(* CODESYS project PacFramwork.project
   Version: 0.0.0.0
   Title: PacFramwork
   Author: roma_mirkevich

Project tree, tasks and I/O mapping:
  PacFramwork : TM241CEC24T/U, Schneider Electric, order no. TM241CEC24T/U, version 5.1.10.10
    application Application
      libraries: SysTimeRtc, * (System); SysTimeCore, * (System); CmpIecTask, * (System); CmpApp, * (System)
      task MAST (freewheeling, priority 15, watchdog 500 ms x 1) calls SR_Main
      program SR_Main [ST]
      global variables SYS
      global variables TEST
      function block PLCFN [ST]
      function TS_PLCFN [ST]
      global variables BUF
      global variables CH
      global variables HMI
      UTD/
        data type PLC_STA
        data type PLC_ALM1
        data type PLS
        data type PLC_CFG
        data type CHBUF
        data type CHCFG
        data type CHHMI
        data type CHSTA
        data type MODULE
        data type SUBMODULE
      CH/
        function CHAIFN [ST]
        function CHAOFN [ST]
        function CHDIFN [ST]
        function CHDOFN [ST]
        function MODULES [ST]
      function INPUT [ST]
      function OUTPUT [ST]
      function ACTUATOR [ST]
      global variables IO
    Ethernet_1 : Ethernet Network, Schneider Electric, version 5.1.10.10
        settings: FTP Server = false
    Serial_Line_1 : Serial line, Schneider Electric, version 5.1.10.10
      Machine_Expert_Network_Manager : Machine Expert-Network Manager, Schneider Electric, version 4.0.0.4
    Serial_Line_2 : Serial line, Schneider Electric, version 5.1.10.10
      Modbus_Manager : Modbus Manager, Schneider Electric, version 4.0.0.4
    CAN_1 : CANopen bus, Schneider Electric, version 5.1.10.10
    DI : Digital Inputs, Schneider Electric, version 5.1.10.10
        input  iwDI_IW0 : WORD  // IW0
        input  ibDI_IB1 : BYTE  // IB1
    DQ : Digital Outputs, Schneider Electric, version 5.1.10.10
        output qwDQ_QW0 : WORD  // QW0
        output qbDQ_QB1 : BYTE  // QB1
    Counters : Counters, Schneider Electric, version 5.1.10.10
    Pulse_Generators : Pulse Generators, Schneider Electric, version 5.1.10.10
    IO_Bus : IO bus - TM3, Schneider Electric, version 5.1.10.10
      Module_2 : TM3DI32K, Schneider Electric, order no. TM3DI32K, version 1.0.2.2
          input  Application.IO.DI[1] : BOOL  // ID0.I0
          input  Application.IO.DI[2] : BOOL  // ID0.I1
          input  Application.IO.DI[3] : BOOL  // ID0.I2
          input  Application.IO.DI[4] : BOOL  // ID0.I3
          input  Application.IO.DI[5] : BOOL  // ID0.I4
          input  Application.IO.DI[6] : BOOL  // ID0.I5
          input  Application.IO.DI[7] : BOOL  // ID0.I6
          input  Application.IO.DI[8] : BOOL  // ID0.I7
          input  Application.IO.DI[9] : BOOL  // ID0.I8
          input  Application.IO.DI[10] : BOOL  // ID0.I9
          input  Application.IO.DI[11] : BOOL  // ID0.I10
          input  Application.IO.DI[12] : BOOL  // ID0.I11
          input  Application.IO.DI[13] : BOOL  // ID0.I12
          input  Application.IO.DI[14] : BOOL  // ID0.I13
          input  Application.IO.DI[15] : BOOL  // ID0.I14
          input  Application.IO.DI[16] : BOOL  // ID0.I15
          input  Application.IO.DI[17] : BOOL  // ID0.I16
          input  Application.IO.DI[18] : BOOL  // ID0.I17
          input  Application.IO.DI[19] : BOOL  // ID0.I18
          input  Application.IO.DI[20] : BOOL  // ID0.I19
          input  Application.IO.DI[21] : BOOL  // ID0.I20
          input  Application.IO.DI[22] : BOOL  // ID0.I21
          input  Application.IO.DI[23] : BOOL  // ID0.I22
          input  Application.IO.DI[24] : BOOL  // ID0.I23
          input  Application.IO.DI[25] : BOOL  // ID0.I24
          input  Application.IO.DI[26] : BOOL  // ID0.I25
          input  Application.IO.DI[27] : BOOL  // ID0.I26
          input  Application.IO.DI[28] : BOOL  // ID0.I27
          input  Application.IO.DI[29] : BOOL  // ID0.I28
          input  Application.IO.DI[30] : BOOL  // ID0.I29
          input  Application.IO.DI[31] : BOOL  // ID0.I30
          input  Application.IO.DI[32] : BOOL  // ID0.I31
          unmapped channels: ID0
      Module_3 : TM3DQ32TK, Schneider Electric, order no. TM3DQ32TK, version 1.0.2.2
          output Application.IO.DQ[1] : BOOL  // QD0.Q0
          output Application.IO.DQ[2] : BOOL  // QD0.Q1
          output Application.IO.DQ[3] : BOOL  // QD0.Q2
          output Application.IO.DQ[4] : BOOL  // QD0.Q3
          output Application.IO.DQ[5] : BOOL  // QD0.Q4
          output Application.IO.DQ[6] : BOOL  // QD0.Q5
          output Application.IO.DQ[7] : BOOL  // QD0.Q6
          output Application.IO.DQ[8] : BOOL  // QD0.Q7
          output Application.IO.DQ[9] : BOOL  // QD0.Q8
          output Application.IO.DQ[10] : BOOL  // QD0.Q9
          output Application.IO.DQ[11] : BOOL  // QD0.Q10
          output Application.IO.DQ[12] : BOOL  // QD0.Q11
          output Application.IO.DQ[13] : BOOL  // QD0.Q12
          output Application.IO.DQ[14] : BOOL  // QD0.Q13
          output Application.IO.DQ[15] : BOOL  // QD0.Q14
          output Application.IO.DQ[16] : BOOL  // QD0.Q15
          output Application.IO.DQ[17] : BOOL  // QD0.Q16
          output Application.IO.DQ[18] : BOOL  // QD0.Q17
          output Application.IO.DQ[19] : BOOL  // QD0.Q18
          output Application.IO.DQ[20] : BOOL  // QD0.Q19
          output Application.IO.DQ[21] : BOOL  // QD0.Q20
          output Application.IO.DQ[22] : BOOL  // QD0.Q21
          output Application.IO.DQ[23] : BOOL  // QD0.Q22
          output Application.IO.DQ[24] : BOOL  // QD0.Q23
          output Application.IO.DQ[25] : BOOL  // QD0.Q24
          output Application.IO.DQ[26] : BOOL  // QD0.Q25
          output Application.IO.DQ[27] : BOOL  // QD0.Q26
          output Application.IO.DQ[28] : BOOL  // QD0.Q27
          output Application.IO.DQ[29] : BOOL  // QD0.Q28
          output Application.IO.DQ[30] : BOOL  // QD0.Q29
          output Application.IO.DQ[31] : BOOL  // QD0.Q30
          output Application.IO.DQ[32] : BOOL  // QD0.Q31
          unmapped channels: QD0
      Module_4 : TM3AI8/G, Schneider Electric, order no. TM3AI8/G, version 1.0.2.2
          input  Application.IO.AI[1] : INT  // IW0
          input  Application.IO.AI[2] : INT  // IW1
          input  Application.IO.AI[3] : INT  // IW2
          input  Application.IO.AI[4] : INT  // IW3
          input  Application.IO.AI[5] : INT  // IW4
          input  Application.IO.AI[6] : INT  // IW5
          input  Application.IO.AI[7] : INT  // IW6
          input  Application.IO.AI[8] : INT  // IW7
          input  ibModule_4_IBStatusIW0 : BYTE  // IBStatusIW0
          input  ibModule_4_IBStatusIW1 : BYTE  // IBStatusIW1
          input  ibModule_4_IBStatusIW2 : BYTE  // IBStatusIW2
          input  ibModule_4_IBStatusIW3 : BYTE  // IBStatusIW3
          input  ibModule_4_IBStatusIW4 : BYTE  // IBStatusIW4
          input  ibModule_4_IBStatusIW5 : BYTE  // IBStatusIW5
          input  ibModule_4_IBStatusIW6 : BYTE  // IBStatusIW6
          input  ibModule_4_IBStatusIW7 : BYTE  // IBStatusIW7
      Module_5 : TM3AQ4/G, Schneider Electric, order no. TM3AQ4/G, version 1.0.2.2
          output Application.IO.AQ[1] : INT  // QW0
          output Application.IO.AQ[2] : INT  // QW1
          output Application.IO.AQ[3] : INT  // QW2
          output Application.IO.AQ[4] : INT  // QW3
          input  ibModule_5_IBStatusQW0 : BYTE  // IBStatusQW0
          input  ibModule_5_IBStatusQW1 : BYTE  // IBStatusQW1
          input  ibModule_5_IBStatusQW2 : BYTE  // IBStatusQW2
          input  ibModule_5_IBStatusQW3 : BYTE  // IBStatusQW3
      Module_6 : TM3AQ4/G, Schneider Electric, order no. TM3AQ4/G, version 1.0.2.2
          output Application.IO.AQ[5] : INT  // QW0
          output Application.IO.AQ[6] : INT  // QW1
          output Application.IO.AQ[7] : INT  // QW2
          output Application.IO.AQ[8] : INT  // QW3
          input  ibModule_6_IBStatusQW0 : BYTE  // IBStatusQW0
          input  ibModule_6_IBStatusQW1 : BYTE  // IBStatusQW1
          input  ibModule_6_IBStatusQW2 : BYTE  // IBStatusQW2
          input  ibModule_6_IBStatusQW3 : BYTE  // IBStatusQW3
    Cartridge_1 : Cartridge, Schneider Electric, version 5.1.10.10
    COM_Bus : COM bus, Schneider Electric, version 5.1.10.10
*)

// PacFramwork/Application/UTD/PLC_STA
TYPE PLC_STA :
STRUCT
      CON2ERR  : BOOL;   // =1 - є помилка звязку з сусідні ПЛК в парі (для теплого резерування)
      PLC2STOP : BOOL;   // =1 - спарений ПЛК в стопі (для теплого резерування)
      BLK  	   : BOOL;   // =1 – є хоча б один заблокований ВМ
      ALDIS    : BOOL; 	 // =1 – є хоча б одна відключена тривога
      DIOON    : BOOL;   // =1 - йде опитування по мережі (MODBUS або аналогічній) засобів віддаленого вводу/виводу
      DIOERR   : BOOL;   // =1 - є помилка на DIO
      b6       : BOOL; 
      FRC      : BOOL;   // =1 – хоча б одна змінна форсована на будь якому рівні
      SMLALL   : BOOL; 	 // =1 – все в режимі в імітації, примушує усі CM перейти в режим імітації
      DISP     : BOOL;   // =1 – хоча б один елемент в режимі ручного управління
      FRC2     : BOOL;   // =1 – є хоча б один форсований керівний елемент (рівня 2), клапан, двигун
      FRC1     : BOOL;   // =1 – хоча б одна змінна форсована (рівня 1)
      SCN1     : BOOL;   // =1 – перший скан
      FRC0     : BOOL;   // =1 – хоча б одна змінна форсована (рівня 0)
      SML      : BOOL;   // =1 – хоча б один об’єкт в режимі імітації
      CMDACK   : BOOL;   // =1 - підтвердження команди, команда пройшла через весь цикл задачі і отримана усіма	
END_STRUCT
END_TYPE

// PacFramwork/Application/UTD/PLC_ALM1
TYPE PLC_ALM1 :
STRUCT
	  ALM      : BOOL;    // =1 - є активна тривога
      NWALM    : BOOL;    // =1 - є нова тривога 
      ALMNACK  : BOOL;    // =1 - біт підтвердження тривоги 
      WRN      : BOOL;    // =1 - є активне попередження
      NWWRN    : BOOL;    // =1 - є нове попередження 
      WRNNACK  : BOOL;    // =1 - біт підтвердження попередження 
      BAD      : BOOL;	  // =1 - є активна тривога недостовірності даних
      NWBAD    : BOOL;	  // =1 - є нова тривога недостовірності даних 
      BADNACK  : BOOL;	  // =1 - біт підтвердження тривоги недостовірності даних 
      EMCYSTP  : BOOL; 	  // =1, аварійний зупин (грибок)
      STP2RUN  : BOOL;    // =1, момент переходу з аварійного зупину в роботу
      CON2ERR  : BOOL;    // =1 - є помилка звязку з сусідні ПЛК в парі (для теплого резерування)
      PLC2STOP : BOOL; 	  // =1 - спарений ПЛК в стопі (для теплого резерування)
      DIOERR   : BOOL;    // =1 - є помилка DIO
      PLCERR   : BOOL;    // =1 – є апаратна помилка (ПЛК)
      CONHIERR : BOOL;    // =1 – єпомилка звязку з верхнім рівнем
END_STRUCT
END_TYPE

// PacFramwork/Application/UTD/PLS
TYPE PLS :
STRUCT
	  P100MS   : BOOL;   // 100 мс
      P200MS   : BOOL;   // 200 мс
      P500MS   : BOOL;   // 500 мс
      P1S      : BOOL;   // 1 с
      P2S      : BOOL;   // 2 с
      P5S      : BOOL;   // 5 с
      P10S     : BOOL;   // 10 с
      P60S     : BOOL;   // 1 хв
      M1S      : BOOL;   // меандр з періодом 1 с (0.5 с + 0.5 с)
      M2S      : BOOL;   // меандр з періодом 2 с (1 с + 1 с)
      b10      : BOOL;
      b11      : BOOL;
      NEWMIN   : BOOL;   // =1 (на один цикл основної задачі) – початок хвилини
      NEWHR    : BOOL;   // =1 (на один цикл основної задачі) – початок години
      NEWDAY   : BOOL;   // =1 (на один цикл основної задачі) – початок доби
      NEWSHIFT : Bool;   // =1 (на один цикл основної задачі) – початок зміни
END_STRUCT
END_TYPE

// PacFramwork/Application/UTD/PLC_CFG
TYPE PLC_CFG :
STRUCT
	  ID          : UINT;                 // Унікальний ідентифікатор
      CLSID       : UINT;                 // 1621xx
      STA         : PLC_STA;              // набір біт типу PLC_STA
      CMD         : UINT;                 // Команди з HMI
      CMDPRG      : UINT;                 // Команди з програмного керування (побітові)
      PRM1        : UINT;                 // дискретні параметри
      PRM2        : UINT;                 // дискретні параметри
      PLS         : PLS;                  // бітові міандри
      ALM1        : PLC_ALM1;             // біти алармів
      ALM2        : INT;                  // біти алармів
      STEP1       : INT;                  // крок основної програми
      T_STEP1     : INT;                  // час кроку основної програми обробки, в (с)
      MSG         : UDINT;                // для формування повідомлень, може бути як бітовим (32 повідомлення), так і числовим (за номером); передбачається, що повідомлення буде скидуватися в 0 автоматично через певний час (не менш ніж 2 інтервали опитування з HMI)
      TQ          : UDINT;                // загальний час з початку 1-го циклу контролера (в секундах)
      TQM         : UDINT;                // загальний час роботи ПЛК з моменту пуску (в хвилинах)
      DICNT       : INT;                  // кількість наявних каналів DI
      DOCNT       : INT;                  // кількість наявних каналів DO
      AICNT       : INT;                  // кількість наявних каналів AI
      AOCNT       : INT;                  // кількість наявних каналів AO
      NOW         : ARRAY[0..3] OF INT;   // плинний час астрономічний час в BCD форматі: NOW[0] seconds,-- (16ss,--)  NOW[1] hour, minute (16hhmm)  NOW[2] month, day (16mmdd)  NOW[3] year (16yyyy)
      SHIFTPARA   : ARRAY[0..3] OF INT;   // Години передачі змін (максимум 3 зміни): SHIFT[0] – кількість змін SHIFT[1] – передача 1-ї зміни (BCD 16hhmm) SHIFT[2] – передача 2-ї зміни (BCD 16hhmm)  SHIFT[3] – передача 3-ї зміни (BCD 16hhmm)
      SHIFTNMB    : UINT;                 // номер активної зміни
      CNTALM      : UINT;                 // лічильник кількості активних тривог аварія
      CNTWRN      : UINT;                 // лічильник кількостіактивних тривог попередження
      CNTBAD      : UINT;                 // лічильник кількостіактивних тривог недостовірність
      CNTFRC      : UINT;                 // лічильник кількостіфорсованих об'єктів
      CNTMAN      : UINT;                 // лічильник кількості ВМ в ручному режимі
      TSK_LTIME   : UINT;                 // плинний (останній) час задачі в мілісекундах
      TSK_MAXTIME : UINT;                 // максимальний час задачі в мілісекундах
      STA_PERM    : UINT;                 // повторює STA, який був на початку виклику функції
      ALM1_PERM   : UINT;                 // повторює ALM1, який був на початку виклику функції
      CNTALM_PERM : UINT := 0;            // лічильник кількості активних тривог аварія
      CNTWRN_PERM : UINT := 0;            // лічильник кількостіактивних тривог попередження
      CNTBAD_PERM : UINT := 0;            // лічильник кількостіактивних тривог недостовірність
      CNTFRC_PERM : UINT := 0;            // лічильник кількостіфорсованих об'єктів
      CNTMAN_PERM : UINT := 0;            // лічильник кількості ВМ в ручному режимі
	  MODULSCNT : INT;   // кількість модулів
      NOWns : UDInt;   // нс (наносекунди) для плинного астрономічного часу 
      TQMS : UDInt;   // мілісекундний лічильник, скидається при старті або після переповнення 
END_STRUCT
END_TYPE

// PacFramwork/Application/UTD/CHBUF
TYPE CHBUF :
STRUCT
ID:	UINT;
CLSID:	UINT;
STA:	INT;
CMD:	INT;
VAL:	INT;
VARID:	UINT;
END_STRUCT
END_TYPE

// PacFramwork/Application/UTD/CHCFG
TYPE CHCFG :
STRUCT
ID:	UINT;
CLSID:	UINT;
STA:	CHSTA;
CMD:	INT;
VAL:	INT;
VARID:	UINT;
END_STRUCT
END_TYPE

// PacFramwork/Application/UTD/CHHMI
TYPE CHHMI :
STRUCT
STA:	INT;
VAL:	INT;
END_STRUCT
END_TYPE

// PacFramwork/Application/UTD/CHSTA
TYPE CHSTA :
STRUCT
VRAW:	BOOL;
VAL:	BOOL;
BAD:	BOOL;
b3:	BOOL;
PNG:	BOOL;
ULNK:	BOOL;
MERR:	BOOL;
BRK:	BOOL;
SHRT:	BOOL;
NBD:	BOOL;
b10:	BOOL;
b11:	BOOL;
INBUF:	BOOL;
FRC:	BOOL;
SML:	BOOL;
CMDLOAD:	BOOL;
END_STRUCT
END_TYPE

// PacFramwork/Application/UTD/MODULE
TYPE MODULE :
STRUCT
STA:	INT;
TYPE1:	INT;
CHCNTS:	INT;
REZ:	INT;
STRTNMB:	ARRAY[0..3] OF INT;
END_STRUCT
END_TYPE

// PacFramwork/Application/UTD/SUBMODULE
TYPE SUBMODULE :
STRUCT
STRTNMB:	INT;
CNT:	INT;
TYPE1:	INT;
CMD:	INT;
CH:	ARRAY[0..15] OF CHHMI;

END_STRUCT
END_TYPE

// PacFramwork/Application/SYS
{attribute 'qualified_only'}
VAR_GLOBAL
END_VAR
VAR_GLOBAL RETAIN
PLCCFG:	PLC_CFG := (DICNT := 32, DOCNT := 32, AICNT := 8, AOCNT := 8);
CHDI:	ARRAY[0..32] OF CHCFG;
CHDO:	ARRAY[0..32] OF CHCFG;
CHAI:	ARRAY[0..8] OF CHCFG;
CHAO:	ARRAY[0..8] OF CHCFG;

END_VAR

// PacFramwork/Application/TEST
{attribute 'qualified_only'}
VAR_GLOBAL
END_VAR
VAR_GLOBAL RETAIN
	TST_CCLS:INT;
	TST_SCN1CLC:INT;
	TST_NBCLC:INT;
	TST_PLSON:BOOL;
	TST_P100MS:INT;
	TST_P200MS:INT;
	TST_P500MS:INT;
	TST_P1S:INT;
	TST_P2S:INT;
	TST_P5S:INT;
	TST_P10S:INT;
	TST_P60S:INT;
	TEST_TQPREV:UDINT;
	TST_CHHRCNT:INT;
	TST_CHDAYCNT:int;
END_VAR

// PacFramwork/Application/BUF
{attribute 'qualified_only'}
VAR_GLOBAL
CHBUF:	CHBUF;
SUBMODULE:	SUBMODULE;

END_VAR

// PacFramwork/Application/CH
{attribute 'qualified_only'}
VAR_GLOBAL
CHDI:	ARRAY[0..32] OF CHHMI;
CHDO:	ARRAY[0..32] OF CHHMI;
CHAI:	ARRAY[0..10] OF CHHMI;
CHAO:	ARRAY[0..6] OF CHHMI;

END_VAR

// PacFramwork/Application/HMI
{attribute 'qualified_only'}
VAR_GLOBAL
	MODULES:	ARRAY[0..15] OF MODULE;
END_VAR

// PacFramwork/Application/IO
{attribute 'qualified_only'}
VAR_GLOBAL
	DI: ARRAY [1..32] OF BOOL;
	DQ: ARRAY [1..32] OF BOOL;
	AI: ARRAY [1..8] OF INT;
	AQ: ARRAY [1..8] OF INT;
END_VAR

// PacFramwork/Application/SR_Main
PROGRAM SR_Main
VAR
PLCFN:PLCFN;
END_VAR

PLCFN(PLC:=SYS.PLCCFG);
MODULES();
INPUT();

ACTUATOR();
OUTPUT();

//TS_PLCFN();

END_PROGRAM

// PacFramwork/Application/PLCFN
FUNCTION_BLOCK PLCFN
   VAR_IN_OUT 
      PLC : PLC_CFG;
   END_VAR
VAR_STAT
      TMBITS_PREV : Int;   // попереднє значення таймерних меандрів
      MEM_RT : LREAL;   // память для вимірювання часу циклу
	  FirstScan : BOOL ;
	  NextScan : BOOL;
	  Clock_10Hz: BOOL;
      Clock_5Hz: BOOL;
      Clock_2Hz: BOOL;
      Clock_1Hz: BOOL;
	  Clock_0_5Hz: BOOL;
	  BLINK_10Hz: BLINK;
	  BLINK_5Hz: BLINK;
	  BLINK_2Hz: BLINK;
	  BLINK_1Hz: BLINK;
	  BLINK_0_5Hz: BLINK;
	  iecResult  :    RTS_IEC_RESULT;
	  pIecInfo   :    POINTER TO CmpIecTask.Task_Info2;
	  LocalTime_ofset:INT:=2;
END_VAR

VAR_TEMP 
      TMBITS_CUR : Int;
      i : INT;
	  NOW: SYSTIMEDATE;
END_VAR

	IF PLC.STA.CMDACK THEN
	    PLC.CMD := 0;
	END_IF;
	PLC.STA.CMDACK := (PLC.CMD <> 0 AND NOT PLC.STA.CMDACK);
	
	(*--------------------------------- Визначення біту першого скану*)
	
	IF NOT FirstScan AND NOT NextScan THEN
		FirstScan := TRUE;
		NextScan:=TRUE;
	ELSE
		FirstScan := FALSE;
	END_IF


	
	PLC.STA.SCN1 := FirstScan;
	IF PLC.STA.SCN1 THEN (*при першому скані*)
	    PLC.ID := 1;             (*Ідентифікатор завжди 1*)
	    PLC.CLSID := 16#2100;    (*Клас завжди 162100*)
	    PLC.TQ := 0;
	    TMBITS_CUR := 0;
	    TMBITS_PREV := 0;
		PLC.TQMS := 0;
	END_IF;
	
	PLC.STA_PERM.0 := PLC.STA.CON2ERR;
	PLC.STA_PERM.1 := PLC.STA.PLC2STOP;
	PLC.STA_PERM.2 := PLC.STA.BLK;
	PLC.STA_PERM.3 := PLC.STA.ALDIS;
	PLC.STA_PERM.4 := PLC.STA.DIOON;
	PLC.STA_PERM.5 := PLC.STA.DIOERR;
	PLC.STA_PERM.6 := PLC.STA.b6;
	PLC.STA_PERM.7 := PLC.STA.FRC;
	PLC.STA_PERM.8 := PLC.STA.SMLALL;
	PLC.STA_PERM.9 := PLC.STA.DISP;
	PLC.STA_PERM.10 := PLC.STA.FRC2;
	PLC.STA_PERM.11 := PLC.STA.FRC1;
	PLC.STA_PERM.12 := PLC.STA.SCN1;
	PLC.STA_PERM.13 := PLC.STA.FRC0;
	PLC.STA_PERM.14 := PLC.STA.SML;
	PLC.STA_PERM.15 := PLC.STA.CMDACK;
	
	PLC.ALM1_PERM.0 := PLC.ALM1.ALM;
	PLC.ALM1_PERM.1 := PLC.ALM1.NWALM;
	PLC.ALM1_PERM.2 := PLC.ALM1.ALMNACK;
	PLC.ALM1_PERM.3 := PLC.ALM1.WRN;
	PLC.ALM1_PERM.4 := PLC.ALM1.NWWRN;
	PLC.ALM1_PERM.5 := PLC.ALM1.WRNNACK;
	PLC.ALM1_PERM.6 := PLC.ALM1.BAD;
	PLC.ALM1_PERM.7 := PLC.ALM1.NWBAD;
	PLC.ALM1_PERM.8 := PLC.ALM1.BADNACK;
	PLC.ALM1_PERM.9 := PLC.ALM1.EMCYSTP;
	PLC.ALM1_PERM.10 := PLC.ALM1.STP2RUN;
	PLC.ALM1_PERM.11 := PLC.ALM1.CON2ERR;
	PLC.ALM1_PERM.12 := PLC.ALM1.PLC2STOP;
	PLC.ALM1_PERM.13 := PLC.ALM1.DIOERR;
	PLC.ALM1_PERM.14 := PLC.ALM1.PLCERR;
	PLC.ALM1_PERM.15 := PLC.ALM1.CONHIERR;
	
	
	(*--------------------------------- таймерні біти та лічильники*)
	BLINK_10Hz(enable:=TRUE, timelow:=T#50MS, timehigh:=T#50MS, out=>Clock_10Hz);
	BLINK_5Hz(enable:=TRUE, timelow:=T#100MS, timehigh:=T#100MS, out=>Clock_5Hz);
	BLINK_2Hz(enable:=TRUE, timelow:=T#250MS, timehigh:=T#250MS, out=>Clock_2Hz);
	BLINK_1Hz(enable:=TRUE, timelow:=T#500MS, timehigh:=T#500MS, out=>Clock_1Hz);
	BLINK_0_5Hz(enable:=TRUE, timelow:=T#1000MS, timehigh:=T#1000MS, out=>Clock_0_5Hz);
	
	(*плинні значення*)
	TMBITS_CUR.0 := Clock_10Hz;         // 100MS 
	TMBITS_CUR.1 := Clock_5Hz;        // 200MS
	TMBITS_CUR.2 := Clock_2Hz;        // 500MS
	TMBITS_CUR.3 := Clock_1Hz;      // 1S
	TMBITS_CUR.7 := PLC.NOW[0] > 16#29; //min
	
	(*відловлювання імпульсів необхідних часових періодів*)
	PLC.PLS.P100MS := TMBITS_CUR.0 AND NOT TMBITS_PREV.0; (*100 мс *)
	PLC.PLS.P200MS := TMBITS_CUR.1 AND NOT TMBITS_PREV.1; (*200 мс*)
	PLC.PLS.P500MS := TMBITS_CUR.2 AND NOT TMBITS_PREV.2; (*500 мс*)
	PLC.PLS.P1S := TMBITS_CUR.3 AND NOT TMBITS_PREV.3; (*1 с*)
	PLC.PLS.P60S := TMBITS_CUR.7 AND NOT TMBITS_PREV.7; (*1 хв*)
	(*підрахунок кількості секунд і хвилин*)
	IF PLC.PLS.P1S THEN
	    PLC.TQ := PLC.TQ + 1;
	END_IF;  (*загальний час з початку 1-го циклу контролера (в секундах)*)
	IF PLC.TQ > 16#7FFF_FFFF THEN
	    PLC.TQ := 16#7FFF_FFFF;
	END_IF;
	IF PLC.PLS.P60S AND NOT PLC.STA.SCN1 THEN
	    PLC.TQM := PLC.TQM + 1;
	END_IF; (*загальний час роботи ПЛК з моменту пуску (в хвилинах)*)
	IF PLC.TQM > 16#7FFF_FFFF THEN
	    PLC.TQM := 16#7FFF_FFFF;
	END_IF;
	
	(*розрахунок інших часових періодів*)
	PLC.PLS.P2S := (PLC.TQ MOD 2) = 0 AND PLC.PLS.P1S;(*2 с*)
	PLC.PLS.P5S := (PLC.TQ MOD 5) = 0 AND PLC.PLS.P1S;(*5 с*)
	PLC.PLS.P10S := (PLC.TQ MOD 10) = 0 AND PLC.PLS.P1S;(*10 с*)
	
	(* меандри *)
	PLC.PLS.M1S := Clock_1Hz;  (*меандр з періодом 1 с (0.5 с + 0.5 с)*)
	PLC.PLS.M2S := Clock_0_5Hz;(*меандр з періодом 2 с (1 с + 1 с) *)
	
	(* астрономічний час *)
	SysTimeRtcConvertUtcToDate(dwTimestampUtc:= GetRTC()+LocalTime_ofset*3600, pDate:=NOW );
	PLC.NOW[0] := INT_TO_BCD(NOW.wSECOND); //NOW[0] seconds,-- (16ss,--)
	PLC.NOW[1] := SHL(INT_TO_BCD(NOW.wHOUR), 8) OR INT_TO_BCD(NOW.wMINUTE);//16hhmm
	PLC.NOW[2] := SHL(INT_TO_BCD(NOW.wMONTH), 8) OR INT_TO_BCD(NOW.wDAY);  //16mmdd
	PLC.NOW[3] := SHL(INT_TO_BCD(NOW.wYEAR / 100), 8) OR INT_TO_BCD(NOW.wYEAR MOD 100);; //16yyyy
	PLC.NOWns := INT_TO_BCD(now.wMilliseconds)*1000000;
	(* початок години *)
	PLC.PLS.NEWHR := (PLC.NOW[1] AND 16#00FF) = 0 (*хвилини*)AND PLC.PLS.P60S (*один раз за хвилину*);
	
	(* початок доби*)
	PLC.PLS.NEWDAY := PLC.NOW[1] = 0 (*години_хвилини*)AND PLC.PLS.P60S (*один раз за хвилину*);
	
	(*початок зміни*)
	IF PLC.SHIFTPARA[0] < 1 OR PLC.SHIFTPARA[0] > 3 THEN
	    PLC.SHIFTPARA[0] := 2;
	END_IF;(*коректність кількості змін*)
	PLC.PLS.NEWSHIFT := FALSE; (*скидуємо біт початку зміни*)
	FOR i := 1 TO PLC.SHIFTPARA[0] DO
	    (*хоча б одна з устоавок змін спрацювала*)
	    PLC.PLS.NEWSHIFT := PLC.PLS.NEWSHIFT OR (PLC.SHIFTPARA[i] = PLC.NOW[1] (*години хвилин*)AND PLC.PLS.P60S (*один раз за хвилину*));
	END_FOR;
	
	TMBITS_PREV := TMBITS_CUR;(*збереження попередніх значень*)
	
	(*----------- визначеня зміни*)
	IF PLC.SHIFTPARA[0] > 3 OR PLC.SHIFTPARA[0] < 2 THEN
	    PLC.SHIFTPARA[0] := 3;
	END_IF;(*якщо кількість змін >3 або <1 - робимо 3*)
	IF PLC.NOW[1] >= PLC.SHIFTPARA[1] AND (PLC.NOW[1] < PLC.SHIFTPARA[2] OR PLC.SHIFTPARA[2] = 16#0000) THEN (*1-ша зміна*)
	    PLC.SHIFTNMB := 1;
	ELSE (*2-га або 3-тя*)
	    IF PLC.SHIFTPARA[0] = 2 THEN (*якщо в 2 зміни*)
	        PLC.SHIFTNMB := 2;
	    ELSE (*якщо 3 зміни*)
	        IF PLC.NOW[1] >= PLC.SHIFTPARA[2] AND (PLC.NOW[1] < PLC.SHIFTPARA[3] OR PLC.SHIFTPARA[3] = 16#0000) THEN
	            PLC.SHIFTNMB := 2;
	        ELSE
	            PLC.SHIFTNMB := 3;
	        END_IF;
	    END_IF;
	END_IF;
	(*----------- *)
	
	(*цикли*)
	pIecInfo := IecTaskGetInfo3(hIecTask := IecTaskGetCurrent(pResult := ADR(iecResult)), pResult := ADR(iecResult));
	PLC.TSK_LTIME := DWORD_TO_UINT(pIecInfo^.dwCycleTime / 1000);
	
	
	IF NOT FirstScan THEN
	    //обмеження 
	    IF PLC.TSK_MAXTIME > 3000 THEN
	        PLC.TSK_MAXTIME := 0;
	    END_IF;
	    IF PLC.TSK_MAXTIME < PLC.TSK_LTIME THEN
	        PLC.TSK_MAXTIME := PLC.TSK_LTIME;
	    END_IF;
	ELSE
	    PLC.TSK_MAXTIME := 0;
	END_IF;
	PLC.TQMS := PLC.TQMS + PLC.TSK_LTIME;//лічильник в мс
	
	(*скидання статусів і тривог*)
	PLC.STA.BLK := false;
	PLC.STA.ALDIS := false;
	PLC.STA.FRC := false;
	PLC.STA.SMLALL := false;
	PLC.STA.DISP := false;
	PLC.STA.FRC2 := false;
	PLC.STA.FRC1 := false;
	PLC.STA.FRC0 := false;
	PLC.STA.SML := false;
	
	PLC.ALM1.ALM := 0;
	PLC.ALM1.NWALM := 0;
	PLC.ALM1.ALMNACK := 0;
	PLC.ALM1.WRN := 0;
	PLC.ALM1.NWWRN := 0;
	PLC.ALM1.WRNNACK := 0;
	PLC.ALM1.BAD := 0;
	PLC.ALM1.NWBAD := 0;
	PLC.ALM1.BADNACK := 0;
	PLC.ALM1.EMCYSTP := 0;
	PLC.ALM1.STP2RUN := 0;
	PLC.ALM1.CON2ERR := 0;
	PLC.ALM1.PLC2STOP := 0;
	PLC.ALM1.DIOERR := 0;
	PLC.ALM1.PLCERR := 0;
	PLC.ALM1.CONHIERR := 0;
	
	(*запамятовування лічильників*)
	PLC.CNTALM_PERM := PLC.CNTALM;
	PLC.CNTWRN_PERM := PLC.CNTWRN;
	PLC.CNTBAD_PERM := PLC.CNTBAD;
	PLC.CNTFRC_PERM := PLC.CNTFRC;
	PLC.CNTMAN_PERM := PLC.CNTMAN;
	
	(*скидання лічильників*)
	PLC.CNTALM := 0;
	PLC.CNTWRN := 0;
	PLC.CNTBAD := 0;
	PLC.CNTFRC := 0;
	PLC.CNTMAN := 0;

END_FUNCTION_BLOCK

// PacFramwork/Application/CH/MODULES
FUNCTION MODULES : BOOL
VAR_INPUT
END_VAR
VAR
i:	INT;
j:	INT;
sbmtype:	INT;
sbmchcnts:	INT;
sbmstrtnmb:	INT;
sbmCMD:	INT;
modtype:	INT;
modchcnts:	INT;
modSTA:	INT;
mask:	INT;
cmdLoadsbm:	BOOL;
cmdLoadch:	BOOL;
sbmbad:	BOOL;
inbuf:	BOOL;
zm:	INT;
k:	INT;

END_VAR

//перебір усіх модулів
FOR i := 0 TO SYS.PLCCFG.MODULSCNT - 1 DO
    modtype := HMI.MODULES[i].TYPE1; //тип модуля
    modchcnts := HMI.MODULES[i].CHCNTS;//кількість каналів в кожному підмодулі
    modSTA := 0; //стан
    //проходження по підмодулям
    FOR j := 0 TO 3 DO
        zm := 12 - 4 * j; //зміщення для SHIFT
        //тип підмодуля
        sbmtype := SHR(modtype, zm) AND 16#000F;
        //кількість каналів у підмодулі
        sbmchcnts := (SHR(modchcnts, zm) AND 16#000F) + 1;
        //початковий індекс каналу 
        sbmstrtnmb := HMI.MODULES[i].STRTNMB[j];
        //перевірка бітових команд
        mask := 16#0800; //маска для зміщення біту команди
        cmdLoadsbm := (HMI.MODULES[i].STA AND SHR(mask, j)) <> 0;
        //завантаження в буфер підмодуля
        IF cmdLoadsbm THEN
            BUF.SUBMODULE.TYPE1 := sbmtype;
            BUF.SUBMODULE.CNT := sbmchcnts;
            BUF.SUBMODULE.STRTNMB := sbmstrtnmb;
        END_IF;
        //визначення помилки на модулі по біту MERR першого каналу в модулі
        CASE sbmtype OF
            1:  //DI
                sbmbad := CH.CHDI[sbmstrtnmb].STA.6; //MERR
            2:  //DQ
                sbmbad := CH.CHDO[sbmstrtnmb].STA.6; //MERR
            3:  //AI
                sbmbad := CH.CHAI[sbmstrtnmb].STA.6; //MERR
            4:  //AO
                sbmbad := CH.CHAO[sbmstrtnmb].STA.6; //MERR
        END_CASE;
        mask := 16#0008; //маска для зміщення біту помилки
        IF sbmbad THEN
            modSTA := modSTA OR SHR(mask, j);
        END_IF;
        //визначення того, що цей підмодуль в буфері  
        inbuf := sbmtype <> 0 AND (BUF.SUBMODULE.TYPE1 = sbmtype) AND (BUF.SUBMODULE.STRTNMB = sbmstrtnmb);
        mask := 16#0080;
        IF inbuf THEN
            modSTA := modSTA OR SHR(mask, j);        END_IF;
        //робота підмодулем в буфері
        IF inbuf THEN
            sbmCMD := BUF.SUBMODULE.CMD;//команда для підмодуля
            //перевірка команди і завантаження значення каналів в буфер 
            FOR k := 0 TO sbmchcnts DO
                cmdLoadch := sbmCMD = k + 1; //завантажити канал
                CASE sbmtype OF
                    16#1:  //DI
                        CH.CHDI[sbmstrtnmb + k].STA.15 := cmdLoadch;
                        BUF.SUBMODULE.CH[k] := CH.CHDI[sbmstrtnmb + k];
                    16#2:  //DQ
                        CH.CHDO[sbmstrtnmb + k].STA.15 := cmdLoadch;
                        BUF.SUBMODULE.CH[k] := CH.CHDO[sbmstrtnmb + k];
                    16#3:  //AI
                        CH.CHAI[sbmstrtnmb + k].STA.15 := cmdLoadch;
                        BUF.SUBMODULE.CH[k] := CH.CHAI[sbmstrtnmb + k];
                    16#4:  //AO
                        CH.CHAO[sbmstrtnmb + k].STA.15 := cmdLoadch;
                        BUF.SUBMODULE.CH[k] := CH.CHAO[sbmstrtnmb + k];
                END_CASE;
            END_FOR;
            BUF.SUBMODULE.CMD := 0;
        END_IF;
    END_FOR;
    
    //запис стану в модуль
    HMI.MODULES[i].STA := modSTA;
    
END_FOR;

END_FUNCTION

// PacFramwork/Application/INPUT
FUNCTION INPUT : BOOL
VAR_INPUT
END_VAR
VAR
	I: INT;
END_VAR

CHDIFN (RAW:=0, CHCFG:=SYS.CHDI[0], CHHMI:=CH.CHDI[0]);
CHAIFN (RAWINT:=0, CHCFG:=SYS.CHAI[0], CHHMI:=CH.CHAI[0]);

FOR i := 1 TO SYS.PLCCFG.DICNT DO
    CHDIFN (RAW:=IO.DI[I], CHCFG:=SYS.CHDI[i], CHHMI:=CH.CHDI[i]);
END_FOR;

FOR i := 1 TO SYS.PLCCFG.AICNT DO
    CHAIFN(RAWINT:=IO.AI[I], CHCFG:=SYS.CHAI[i], CHHMI:=CH.CHAI[i]);
END_FOR;

END_FUNCTION

// PacFramwork/Application/CH/CHDIFN
FUNCTION CHDIFN : BOOL
VAR_INPUT
	RAW:	BOOL;
END_VAR
VAR_IN_OUT
	CHCFG:	CHCFG;
	CHHMI:	CHHMI;
END_VAR
VAR
STA:	CHSTA;
STAINT:	INT;
CMD:	INT;
INBUF:	BOOL;
ULNK:	BOOL;
MERR:	BOOL;
BRK:	BOOL;
SHRT:	BOOL;
SML:	BOOL;
FRC:	BOOL;
BAD:	BOOL;
VRAW:	BOOL;
VAL:	BOOL;
PNG:	BOOL;
NBD:	BOOL;
CMDLOAD:	BOOL;

END_VAR

STA := CHCFG.STA;
CMD := CHCFG.CMD;
(*розпаковка з STA*)
VRAW := STA.VRAW;
VAL := STA.VAL;
BAD := STA.BAD;(*керується ззовні*)
PNG := STA.PNG;
ULNK := STA.ULNK;
MERR := STA.MERR;(*керується ззовні*)
BRK := STA.BRK;(*керується ззовні*)
SHRT := STA.SHRT;(*керується ззовні*)
NBD := STA.NBD;(*керується ззовні*)
INBUF := STA.INBUF;
FRC := STA.FRC;
SML := STA.SML;
CMDLOAD := STA.CMDLOAD; (*керується бітом*)

INBUF := (CHCFG.ID = BUF.CHBUF.ID) AND (CHCFG.CLSID = BUF.CHBUF.CLSID);
CMDLOAD := CHHMI.STA.15;
CMD := 0;

(* обробник команд*)
(* широкомовне форсування/дефорсування*) 
IF SYS.PLCCFG.CMD = 16#4301 THEN
    FRC := true; (*форсувати один/усі об'єкти типу*)
END_IF;
IF SYS.PLCCFG.CMD = 16#4302 THEN
    FRC := false; (*дефорсувати об'єкт типу*)
END_IF;
(*вибір джерела команди згідно пріоритету*)
IF CMDLOAD THEN (*з HMI CMDLOAD*)
    CMD := 16#0100;  // записати в буфер
ELSIF INBUF AND BUF.CHBUF.CMD <> 0 THEN (*з буферу*)
    CMD := BUF.CHBUF.CMD;
ELSIF CHCFG.CMD <> 0 THEN
    CMD := CHCFG.CMD;
END_IF;
(*commands*)
CASE CMD OF
    16#1: (*записати 1*)
        IF FRC AND INBUF THEN
            BUF.CHBUF.VAL := 1;
        END_IF;
    16#2: (*записати 0*)
        IF FRC AND INBUF THEN
            BUF.CHBUF.VAL := 0;
        END_IF;
    16#3: (*TOGGLE*)
        IF FRC AND INBUF THEN
            IF VAL THEN
                BUF.CHBUF.VAL := 0;
            ELSE
                BUF.CHBUF.VAL := 1;
            END_IF;
        END_IF;
    16#0100: (*прочитати конфігурацію в буфер*)
        BUF.CHBUF.ID := CHCFG.ID;
        BUF.CHBUF.CLSID := CHCFG.CLSID;
        
        BUF.CHBUF.STA.0 := CHCFG.STA.VRAW;
        BUF.CHBUF.STA.1 := CHCFG.STA.VAL;
        BUF.CHBUF.STA.2 := CHCFG.STA.BAD;
        BUF.CHBUF.STA.3 := CHCFG.STA.b3;
        BUF.CHBUF.STA.4 := CHCFG.STA.PNG;
        BUF.CHBUF.STA.5 := CHCFG.STA.ULNK;
        BUF.CHBUF.STA.6 := CHCFG.STA.MERR;
        BUF.CHBUF.STA.7 := CHCFG.STA.BRK;
        BUF.CHBUF.STA.8 := CHCFG.STA.SHRT;
        BUF.CHBUF.STA.9 := CHCFG.STA.NBD;
        BUF.CHBUF.STA.10 := CHCFG.STA.b10;
        BUF.CHBUF.STA.11 := CHCFG.STA.b11;
        BUF.CHBUF.STA.12 := CHCFG.STA.INBUF;
        BUF.CHBUF.STA.13 := CHCFG.STA.FRC;
        BUF.CHBUF.STA.14 := CHCFG.STA.SML;
        BUF.CHBUF.STA.15 := CHCFG.STA.CMDLOAD;
        
        BUF.CHBUF.VAL := CHCFG.VAL;
        BUF.CHBUF.VARID := CHCFG.VARID;
    16#0300: (*перемкнути форсування*)
        FRC := NOT FRC;
    16#0301: (*форсувати один/усі об'єкти типу*)
        FRC := true;
    16#0302: (*дефорсувати один/усі об'єкти типу*)
        FRC := false;
END_CASE;

(*запис значення змінної*)
IF FRC AND INBUF THEN (*режим форсування з занятим буфером*)
    CHCFG.VAL := BOOL_TO_INT(BUF.CHBUF.VAL > 0);
    VAL := CHCFG.VAL > 0.5;
ELSIF FRC AND NOT INBUF THEN (*режим форсування без занятого буферу*)
    ;(*без змін*)
ELSIF NOT FRC THEN (*не режим форсування*)
    VAL := RAW;
    IF RAW THEN
        CHCFG.VAL := 1;
    ELSE
        CHCFG.VAL := 0;
    END_IF;
END_IF;

(*ping-pong*)
ULNK := PNG; (*прийшов ping - є звязок з верхнім рівнем*)
PNG := false; (*скидання біту PNG звязку з врехнім рівнем PONG*)
IF NOT ULNK THEN
    CHCFG.VARID := 0;
END_IF;

(*скидання оброблених команд*)
CMDLOAD := 0;
CMD := 0;


(*загальносистемні біти та лічильники*)
IF FRC THEN
    SYS.PLCCFG.STA.FRC0 := true;
    SYS.PLCCFG.CNTFRC := SYS.PLCCFG.CNTFRC + 1;
END_IF;

(*упковка в STA*)
STA.VRAW := RAW;
STA.VAL := VAL;
STA.BAD := BAD;(*керується ззовні*)
STA.PNG := PNG;
STA.ULNK := ULNK;
STA.MERR := MERR;(*керується ззовні*)
STA.BRK := BRK;(*керується ззовні*)
STA.SHRT := SHRT;(*керується ззовні*)
STA.NBD := NBD;(*керується ззовні*)
STA.INBUF := INBUF;
STA.FRC := FRC;
STA.SML := SML;
STA.CMDLOAD := CMDLOAD; (*керується бітом*)

CHCFG.STA := STA;
CHCFG.CMD := CMD;

(*упаковка в INT*)
STAINT.0 := VRAW;
STAINT.1 := VAL;
STAINT.2 := BAD;
//STAINT.3 := b3;
STAINT.4 := PNG;
STAINT.5 := ULNK;
STAINT.6 := MERR;
STAINT.7 := BRK;
STAINT.8 := SHRT;
STAINT.9 := NBD;
//STAINT.10 := STA.b10;
//STAINT.11 := STA.b11;
STAINT.12 := INBUF;
STAINT.13 := FRC;
STAINT.14 := SML;
STAINT.15 := FALSE;

CHHMI.STA := STAINT;
CHHMI.VAL := CHCFG.VAL;

(*оновлення буферу*)
IF INBUF THEN
    BUF.CHBUF.STA := STAINT;
    BUF.CHBUF.VARID := CHCFG.VARID;
    BUF.CHBUF.CMD := 0;
    IF NOT FRC THEN
        BUF.CHBUF.VAL := CHCFG.VAL;
    END_IF;
END_IF;

END_FUNCTION

// PacFramwork/Application/CH/CHAIFN
FUNCTION CHAIFN : BOOL
VAR_INPUT
	RAWINT: INT;
END_VAR

VAR_IN_OUT
CHCFG:	CHCFG;
CHHMI:	CHHMI;
END_VAR

VAR
STA:	CHSTA;
STAINT:	INT;
CMD:	INT;
INBUF:	BOOL;
ULNK:	BOOL;
MERR:	BOOL;
BRK:	BOOL;
SHRT:	BOOL;
SML:	BOOL;
FRC:	BOOL;
BAD:	BOOL;
VRAW:	BOOL;
VAL:	BOOL;
PNG:	BOOL;
NBD:	BOOL;
CMDLOAD:	BOOL;

END_VAR
VAR CONSTANT
MIN1:	INT	:=0;
MAX1:	INT :=27648;
MIDLE:	INT :=13824;

END_VAR

STA := CHCFG.STA;
CMD := CHCFG.CMD;
(*розпаковка з STA*)
VRAW := STA.VRAW;
VAL := STA.VAL;
BAD := STA.BAD;(*керується ззовні*)
PNG := STA.PNG;
ULNK := STA.ULNK;
MERR := STA.MERR;(*керується ззовні*)
BRK := STA.BRK;(*керується ззовні*)
SHRT := STA.SHRT;(*керується ззовні*)
NBD := STA.NBD;(*керується ззовні*)
INBUF := STA.INBUF;
FRC := STA.FRC;
SML := STA.SML;
CMDLOAD := STA.CMDLOAD; (*керується бітом*)

INBUF := (CHCFG.ID = BUF.CHBUF.ID) AND (CHCFG.CLSID = BUF.CHBUF.CLSID);
CMDLOAD := CHHMI.STA.15;
CMD := 0;

(* обробник команд*)
(* широкомовне форсування/дефорсування*) 
IF SYS.PLCCFG.CMD = 16#4301 THEN
    FRC := TRUE; (*форсувати один/усі об'єкти типу*)
END_IF;
IF SYS.PLCCFG.CMD = 16#4302 THEN
    FRC := FALSE; (*дефорсувати об'єкт типу*)
END_IF;
(*вибір джерела команди згідно пріоритету*)
IF CMDLOAD THEN (*з HMI CMDLOAD*)
    CMD := 16#0100;  // записати в буфер
ELSIF INBUF AND BUF.CHBUF.CMD <> 0 THEN (*з буферу*)
    CMD := BUF.CHBUF.CMD;
ELSIF CHCFG.CMD <> 0 THEN
    CMD := CHCFG.CMD;
END_IF;
(*commands*)
CASE CMD OF
    16#1: (*записати MAX*)
        IF FRC AND INBUF THEN
            BUF.CHBUF.VAL := MAX1;
        END_IF;
    16#2: (*записати MIN*)
        IF FRC AND INBUF THEN
            BUF.CHBUF.VAL := MIN1;
        END_IF;
    16#3: (*TOGGLE*)
        IF FRC AND INBUF THEN
            BUF.CHBUF.VAL := MIDLE;
        END_IF;
    16#0100: (*прочитати конфігурацію в буфер*)
        BUF.CHBUF.ID := CHCFG.ID;
        BUF.CHBUF.CLSID := CHCFG.CLSID;
        
        BUF.CHBUF.STA.0 := CHCFG.STA.VRAW;
        BUF.CHBUF.STA.1 := CHCFG.STA.VAL;
        BUF.CHBUF.STA.2 := CHCFG.STA.BAD;
        BUF.CHBUF.STA.3 := CHCFG.STA.b3;
        BUF.CHBUF.STA.4 := CHCFG.STA.PNG;
        BUF.CHBUF.STA.5 := CHCFG.STA.ULNK;
        BUF.CHBUF.STA.6 := CHCFG.STA.MERR;
        BUF.CHBUF.STA.7 := CHCFG.STA.BRK;
        BUF.CHBUF.STA.8 := CHCFG.STA.SHRT;
        BUF.CHBUF.STA.9 := CHCFG.STA.NBD;
        BUF.CHBUF.STA.10 := CHCFG.STA.b10;
        BUF.CHBUF.STA.11 := CHCFG.STA.b11;
        BUF.CHBUF.STA.12 := CHCFG.STA.INBUF;
        BUF.CHBUF.STA.13 := CHCFG.STA.FRC;
        BUF.CHBUF.STA.14 := CHCFG.STA.SML;
        BUF.CHBUF.STA.15 := CHCFG.STA.CMDLOAD;
        
        BUF.CHBUF.VAL := CHCFG.VAL;
        BUF.CHBUF.VARID := CHCFG.VARID;
    16#0300: (*перемкнути форсування*)
        FRC := NOT FRC;
    16#0301: (*форсувати один/усі об'єкти типу*)
        FRC := TRUE;
    16#0302: (*дефорсувати один/усі об'єкти типу*)
        FRC := FALSE;
END_CASE;

(*запис значення змінної*)
IF FRC AND INBUF THEN (*режим форсування з занятим буфером*)
    CHCFG.VAL := BUF.CHBUF.VAL;
ELSIF FRC AND NOT INBUF THEN (*режим форсування без занятого буферу*)
    ;(*без змін*)
ELSIF NOT FRC THEN (*не режим форсування*)
    CHCFG.VAL := RAWINT;
END_IF;

(*ping-pong*)
ULNK := PNG; (*прийшов ping - є звязок з верхнім рівнем*)
PNG := FALSE; (*скидання біту PNG звязку з врехнім рівнем PONG*)
IF NOT ULNK THEN
    CHCFG.VARID := 0;
END_IF;

(*скидання оброблених команд*)
CMDLOAD := 0;
CMD := 0;

(*загальносистемні біти та лічильники*)
IF FRC THEN
    SYS.PLCCFG.STA.FRC0 := TRUE;
    SYS.PLCCFG.CNTFRC := SYS.PLCCFG.CNTFRC + 1;
END_IF;


(*упковка в STA*)
STA.VRAW := RAWINT > 0;
STA.VAL := CHCFG.VAL > 0;
STA.BAD := BAD;(*керується ззовні*)
STA.PNG := PNG;
STA.ULNK := ULNK;
STA.MERR := MERR;(*керується ззовні*)
STA.BRK := BRK;(*керується ззовні*)
STA.SHRT := SHRT;(*керується ззовні*)
STA.NBD := NBD;(*керується ззовні*)
STA.INBUF := INBUF;
STA.FRC := FRC;
STA.SML := SML;
STA.CMDLOAD := CMDLOAD; (*керується бітом*)

CHCFG.STA := STA;
CHCFG.CMD := CMD;

(*упаковка в INT*)
STAINT.0 := VRAW;
STAINT.1 := VAL;
STAINT.2 := BAD;
//STAINT.3 := b3;
STAINT.4 := PNG;
STAINT.5 := ULNK;
STAINT.6 := MERR;
STAINT.7 := BRK;
STAINT.8 := SHRT;
STAINT.9 := NBD;
//STAINT.10 := STA.b10;
//STAINT.11 := STA.b11;
STAINT.12 := INBUF;
STAINT.13 := FRC;
STAINT.14 := SML;
STAINT.15 := FALSE;

CHHMI.STA := STAINT;
CHHMI.VAL := CHCFG.VAL;

(*оновлення буферу*)
IF INBUF THEN
    BUF.CHBUF.STA := STAINT;
    BUF.CHBUF.VARID := CHCFG.VARID;
    BUF.CHBUF.CMD := 0;
    IF NOT FRC THEN
        BUF.CHBUF.VAL := CHCFG.VAL;
    END_IF;
END_IF;

END_FUNCTION

// PacFramwork/Application/ACTUATOR
FUNCTION ACTUATOR : BOOL
VAR_INPUT
END_VAR
VAR
END_VAR

END_FUNCTION

// PacFramwork/Application/OUTPUT
FUNCTION OUTPUT : BOOL
VAR_INPUT
END_VAR
VAR
	temp_bool: BOOL;
	temp_int: int;
	i: int;
END_VAR

CHDOFN(RAW=>temp_bool, CHCFG:=SYS.CHDO[0], CHHMI:=CH.CHDO[0]);
CHAOFN(RAWINT=>temp_int, CHCFG:=SYS.CHAO[0], CHHMI:=CH.CHAO[0]);

FOR i := 1 TO SYS.PLCCFG.DOCNT DO
    CHDOFN(RAW=>IO.DQ[i], CHCFG:=SYS.CHDO[i], CHHMI:=CH.CHDO[i]);
END_FOR;

FOR i := 1 TO SYS.PLCCFG.AOCNT DO
    CHAOFN(RAWINT=>IO.AQ[i], CHCFG:=SYS.CHAO[i], CHHMI:=CH.CHAO[i]);
END_FOR;

END_FUNCTION

// PacFramwork/Application/CH/CHDOFN
FUNCTION CHDOFN : BOOL
VAR_OUTPUT
	RAW:	BOOL;
END_VAR
VAR_IN_OUT
	CHCFG:	CHCFG;
	CHHMI:	CHHMI;
END_VAR
VAR
STA:	CHSTA;
STAINT:	INT;
CMD:	INT;
INBUF:	BOOL;
ULNK:	BOOL;
MERR:	BOOL;
BRK:	BOOL;
SHRT:	BOOL;
SML:	BOOL;
FRC:	BOOL;
BAD:	BOOL;
VRAW:	BOOL;
VAL:	BOOL;
PNG:	BOOL;
NBD:	BOOL;
CMDLOAD:	BOOL;

END_VAR

STA := CHCFG.STA;
CMD := CHCFG.CMD;
(*розпаковка з STA*)
VRAW := STA.VRAW;
VAL := STA.VAL;
BAD := STA.BAD;(*керується ззовні*)
PNG := STA.PNG;
ULNK := STA.ULNK;
MERR := STA.MERR;(*керується ззовні*)
BRK := STA.BRK;(*керується ззовні*)
SHRT := STA.SHRT;(*керується ззовні*)
NBD := STA.NBD;(*керується ззовні*)
INBUF := STA.INBUF;
FRC := STA.FRC;
SML := STA.SML;
CMDLOAD := STA.CMDLOAD; (*керується бітом*)

INBUF := (CHCFG.ID = BUF.CHBUF.ID) AND (CHCFG.CLSID = BUF.CHBUF.CLSID);
CMDLOAD := CHHMI.STA.15;
CMD := 0;

(* обробник команд*)
(* широкомовне форсування/дефорсування*) 
IF SYS.PLCCFG.CMD = 16#4301 THEN
    FRC := true; (*форсувати один/усі об'єкти типу*)
END_IF;
IF SYS.PLCCFG.CMD = 16#4302 THEN
    FRC := false; (*дефорсувати об'єкт типу*)
END_IF;
(*вибір джерела команди згідно пріоритету*)
IF CMDLOAD THEN (*з HMI CMDLOAD*)
    CMD := 16#0100;  // записати в буфер
ELSIF INBUF AND BUF.CHBUF.CMD <> 0 THEN (*з буферу*)
    CMD := BUF.CHBUF.CMD;
ELSIF CHCFG.CMD <> 0 THEN
    CMD := CHCFG.CMD;
END_IF;
(*commands*)
CASE CMD OF
    16#1: (*записати 1*)
        IF FRC AND INBUF THEN
            BUF.CHBUF.VAL := 1;
        END_IF;
    16#2: (*записати 0*)
        IF FRC AND INBUF THEN
            BUF.CHBUF.VAL := 0;
        END_IF;
    16#3: (*TOGGLE*)
        IF FRC AND INBUF THEN
            IF VRAW THEN
                BUF.CHBUF.VAL := 0;
            ELSE
                BUF.CHBUF.VAL := 1;
            END_IF;
        END_IF;
    16#0100: (*прочитати конфігурацію в буфер*)
        BUF.CHBUF.ID := CHCFG.ID;
        BUF.CHBUF.CLSID := CHCFG.CLSID;
        
        BUF.CHBUF.STA.0 := CHCFG.STA.VRAW;
        BUF.CHBUF.STA.1 := CHCFG.STA.VAL;
        BUF.CHBUF.STA.2 := CHCFG.STA.BAD;
        BUF.CHBUF.STA.3 := CHCFG.STA.b3;
        BUF.CHBUF.STA.4 := CHCFG.STA.PNG;
        BUF.CHBUF.STA.5 := CHCFG.STA.ULNK;
        BUF.CHBUF.STA.6 := CHCFG.STA.MERR;
        BUF.CHBUF.STA.7 := CHCFG.STA.BRK;
        BUF.CHBUF.STA.8 := CHCFG.STA.SHRT;
        BUF.CHBUF.STA.9 := CHCFG.STA.NBD;
        BUF.CHBUF.STA.10 := CHCFG.STA.b10;
        BUF.CHBUF.STA.11 := CHCFG.STA.b11;
        BUF.CHBUF.STA.12 := CHCFG.STA.INBUF;
        BUF.CHBUF.STA.13 := CHCFG.STA.FRC;
        BUF.CHBUF.STA.14 := CHCFG.STA.SML;
        BUF.CHBUF.STA.15 := CHCFG.STA.CMDLOAD;
        
        BUF.CHBUF.VAL := CHCFG.VAL;
        BUF.CHBUF.VARID := CHCFG.VARID;
    16#0300: (*перемкнути форсування*)
        FRC := NOT FRC;
    16#0301: (*форсувати один/усі об'єкти типу*)
        FRC := true;
    16#0302: (*дефорсувати один/усі об'єкти типу*)
        FRC := false;
END_CASE;

(*запис значення змінної*)
IF FRC AND INBUF THEN (*режим форсування з занятим буфером*)
    CHCFG.VAL := BOOL_TO_INT(BUF.CHBUF.VAL > 0);
    VRAW := CHCFG.VAL > 0.5;
ELSIF FRC AND NOT INBUF THEN (*режим форсування без занятого буферу*)
    ;(*без змін*)
ELSIF NOT FRC THEN (*не режим форсування*)
    VRAW := VAL;
    IF VAL THEN
        CHCFG.VAL := 1;
    ELSE
        CHCFG.VAL := 0;
    END_IF;
END_IF;
RAW := VRAW; (*відправляємо на вихід*)

(*ping-pong*)
ULNK := PNG; (*прийшов ping - є звязок з верхнім рівнем*)
PNG := false; (*скидання біту PNG звязку з врехнім рівнем PONG*)
IF NOT ULNK THEN
    CHCFG.VARID := 0;
END_IF;

(*скидання оброблених команд*)
CMDLOAD := 0;
CMD := 0;


(*загальносистемні біти та лічильники*)
IF FRC THEN
    SYS.PLCCFG.STA.FRC0 := true;
    SYS.PLCCFG.CNTFRC := SYS.PLCCFG.CNTFRC + 1;
END_IF;

(*упковка в STA*)
STA.VRAW := VRAW;
STA.VAL := VAL;
STA.BAD := BAD;(*керується ззовні*)
STA.PNG := PNG;
STA.ULNK := ULNK;
STA.MERR := MERR;(*керується ззовні*)
STA.BRK := BRK;(*керується ззовні*)
STA.SHRT := SHRT;(*керується ззовні*)
STA.NBD := NBD;(*керується ззовні*)
STA.INBUF := INBUF;
STA.FRC := FRC;
STA.SML := SML;
STA.CMDLOAD := CMDLOAD; (*керується бітом*)

CHCFG.STA := STA;
CHCFG.CMD := CMD;

(*упаковка в INT*)
STAINT.0 := VRAW;
STAINT.1 := VAL;
STAINT.2 := BAD;
//STAINT.3 := b3;
STAINT.4 := PNG;
STAINT.5 := ULNK;
STAINT.6 := MERR;
STAINT.7 := BRK;
STAINT.8 := SHRT;
STAINT.9 := NBD;
//STAINT.10 := STA.b10;
//STAINT.11 := STA.b11;
STAINT.12 := INBUF;
STAINT.13 := FRC;
STAINT.14 := SML;
STAINT.15 := FALSE;

CHHMI.STA := STAINT;
CHHMI.VAL := CHCFG.VAL;

(*оновлення буферу*)
IF INBUF THEN
    BUF.CHBUF.STA := STAINT;
    BUF.CHBUF.VARID := CHCFG.VARID;
    BUF.CHBUF.CMD := 0;
    IF NOT FRC THEN
        BUF.CHBUF.VAL := CHCFG.VAL;
    END_IF;
END_IF;

END_FUNCTION

// PacFramwork/Application/CH/CHAOFN
FUNCTION CHAOFN : BOOL
VAR_OUTPUT
	RAWINT:	INT;
END_VAR
VAR_IN_OUT
	CHCFG:	CHCFG;
	CHHMI:	CHHMI;
END_VAR
VAR
	STA:	CHSTA;
	STAINT:	INT;
	CMD:	INT;
	INBUF:	BOOL;
	ULNK:	BOOL;
	MERR:	BOOL;
	BRK:	BOOL;
	SHRT:	BOOL;
	SML:	BOOL;
	FRC:	BOOL;
	BAD:	BOOL;
	VRAW:	BOOL;
	VAL:	BOOL;
	PNG:	BOOL;
	NBD:	BOOL;
	CMDLOAD:	BOOL;

END_VAR
VAR CONSTANT
	MIN1:	INT	:=0;
	MAX1:	INT :=	27648;
	MIDLE:	INT :=	13824;

END_VAR

STA := CHCFG.STA;
CMD := CHCFG.CMD;
(*розпаковка з STA*)
VRAW := STA.VRAW;
VAL := STA.VAL;
BAD := STA.BAD;(*керується ззовні*)
PNG := STA.PNG;
ULNK := STA.ULNK;
MERR := STA.MERR;(*керується ззовні*)
BRK := STA.BRK;(*керується ззовні*)
SHRT := STA.SHRT;(*керується ззовні*)
NBD := STA.NBD;(*керується ззовні*)
INBUF := STA.INBUF;
FRC := STA.FRC;
SML := STA.SML;
CMDLOAD := STA.CMDLOAD; (*керується бітом*)

INBUF := (CHCFG.ID = BUF.CHBUF.ID) AND (CHCFG.CLSID = BUF.CHBUF.CLSID);
CMDLOAD := CHHMI.STA.15;
CMD := 0;

(* обробник команд*)
(* широкомовне форсування/дефорсування*) 
IF SYS.PLCCFG.CMD = 16#4301 THEN
    FRC := TRUE; (*форсувати один/усі об'єкти типу*)
END_IF;
IF SYS.PLCCFG.CMD = 16#4302 THEN
    FRC := FALSE; (*дефорсувати об'єкт типу*)
END_IF;
(*вибір джерела команди згідно пріоритету*)
IF CMDLOAD THEN (*з HMI CMDLOAD*)
    CMD := 16#0100;  // записати в буфер
ELSIF INBUF AND BUF.CHBUF.CMD <> 0 THEN (*з буферу*)
    CMD := BUF.CHBUF.CMD;
ELSIF CHCFG.CMD <> 0 THEN
    CMD := CHCFG.CMD;
END_IF;
(*commands*)
CASE CMD OF
    16#1: (*записати MAX*)
        IF FRC AND INBUF THEN
            RAWINT := MAX1;
        END_IF;
    16#2: (*записати MIN*)
        IF FRC AND INBUF THEN
            RAWINT := MIN1;
        END_IF;
    16#3: (*TOGGLE*)
        IF FRC AND INBUF THEN
            RAWINT := MIDLE;
        END_IF;
    16#0100: (*прочитати конфігурацію в буфер*)
        BUF.CHBUF.ID := CHCFG.ID;
        BUF.CHBUF.CLSID := CHCFG.CLSID;
        
        BUF.CHBUF.STA.0 := CHCFG.STA.VRAW;
        BUF.CHBUF.STA.1 := CHCFG.STA.VAL;
        BUF.CHBUF.STA.2 := CHCFG.STA.BAD;
        BUF.CHBUF.STA.3 := CHCFG.STA.b3;
        BUF.CHBUF.STA.4 := CHCFG.STA.PNG;
        BUF.CHBUF.STA.5 := CHCFG.STA.ULNK;
        BUF.CHBUF.STA.6 := CHCFG.STA.MERR;
        BUF.CHBUF.STA.7 := CHCFG.STA.BRK;
        BUF.CHBUF.STA.8 := CHCFG.STA.SHRT;
        BUF.CHBUF.STA.9 := CHCFG.STA.NBD;
        BUF.CHBUF.STA.10 := CHCFG.STA.b10;
        BUF.CHBUF.STA.11 := CHCFG.STA.b11;
        BUF.CHBUF.STA.12 := CHCFG.STA.INBUF;
        BUF.CHBUF.STA.13 := CHCFG.STA.FRC;
        BUF.CHBUF.STA.14 := CHCFG.STA.SML;
        BUF.CHBUF.STA.15 := CHCFG.STA.CMDLOAD;
        
        BUF.CHBUF.VAL := CHCFG.VAL;
        BUF.CHBUF.VARID := CHCFG.VARID;
    16#0300: (*перемкнути форсування*)
        FRC := NOT FRC;
    16#301: (*форсувати один/усі об'єкти типу*)
        FRC := TRUE;
    16#302: (*дефорсувати один/усі об'єкти типу*)
        FRC := FALSE;
END_CASE;

(*запис значення змінної*)
IF FRC AND INBUF THEN (*режим форсування з занятим буфером*)
    RAWINT := BUF.CHBUF.VAL;
ELSIF FRC AND NOT INBUF THEN (*режим форсування без занятого буферу*)
    ;(*без змін*)
ELSIF NOT FRC THEN (*не режим форсування*)
    RAWINT := CHCFG.VAL;
END_IF;

(*ping-pong*)
ULNK := PNG; (*прийшов ping - є звязок з верхнім рівнем*)
PNG := FALSE; (*скидання біту PNG звязку з врехнім рівнем PONG*)
IF NOT ULNK THEN
    CHCFG.VARID := 0;
END_IF;

(*скидання оброблених команд*)
CMDLOAD := 0;
CMD := 0;

(*загальносистемні біти та лічильники*)
IF FRC THEN
    SYS.PLCCFG.STA.FRC0 := TRUE;
    SYS.PLCCFG.CNTFRC := SYS.PLCCFG.CNTFRC + 1;
END_IF;


(*упковка в STA*)
STA.VRAW := RAWINT > 0;
STA.VAL := CHCFG.VAL > 0;
STA.BAD := BAD;(*керується ззовні*)
STA.PNG := PNG;
STA.ULNK := ULNK;
STA.MERR := MERR;(*керується ззовні*)
STA.BRK := BRK;(*керується ззовні*)
STA.SHRT := SHRT;(*керується ззовні*)
STA.NBD := NBD;(*керується ззовні*)
STA.INBUF := INBUF;
STA.FRC := FRC;
STA.SML := SML;
STA.CMDLOAD := CMDLOAD; (*керується бітом*)

CHCFG.STA := STA;
CHCFG.CMD := CMD;

(*упаковка в INT*)
STAINT.0 := VRAW;
STAINT.1 := VAL;
STAINT.2 := BAD;
//STAINT.3 := b3;
STAINT.4 := PNG;
STAINT.5 := ULNK;
STAINT.6 := MERR;
STAINT.7 := BRK;
STAINT.8 := SHRT;
STAINT.9 := NBD;
//STAINT.10 := STA.b10;
//STAINT.11 := STA.b11;
STAINT.12 := INBUF;
STAINT.13 := FRC;
STAINT.14 := SML;
STAINT.15 := FALSE;

CHHMI.STA := STAINT;
CHHMI.VAL := CHCFG.VAL;

(*оновлення буферу*)
IF INBUF THEN
    BUF.CHBUF.STA := STAINT;
    BUF.CHBUF.VARID := CHCFG.VARID;
    BUF.CHBUF.CMD := 0;
    IF NOT FRC THEN
        BUF.CHBUF.VAL := CHCFG.VAL;
    END_IF;
END_IF;

END_FUNCTION

// PacFramwork/Application/TS_PLCFN
FUNCTION TS_PLCFN : BOOL
VAR_INPUT
END_VAR
VAR
END_VAR

TEST.TST_CCLS := TEST.TST_CCLS + 1;
IF SYS.PLCCFG.STA.SCN1 THEN
   TEST.TST_SCN1CLC := TEST.TST_SCN1CLC + 1;
   TEST.TST_NBCLC := TEST.TST_CCLS;
END_IF;

IF TEST.TST_PLSON THEN
    IF SYS.PLCCFG.PLS.P100MS THEN
        TEST.TST_P100MS := TEST.TST_P100MS + 1;
    END_IF;
    IF SYS.PLCCFG.PLS.P200MS THEN
        TEST.TST_P200MS := TEST.TST_P200MS + 1;
    END_IF;
    IF SYS.PLCCFG.PLS.P500MS THEN
        TEST.TST_P500MS := TEST.TST_P500MS + 1;
    END_IF;
    IF SYS.PLCCFG.PLS.P1S THEN
        TEST.TST_P1S := TEST.TST_P1S + 1;
    END_IF;
    IF SYS.PLCCFG.PLS.P2S THEN
        TEST.TST_P2S := TEST.TST_P2S + 1;
    END_IF;
    IF SYS.PLCCFG.PLS.P5S THEN
        TEST.TST_P5S := TEST.TST_P5S + 1;
    END_IF;
    IF SYS.PLCCFG.PLS.P10S THEN
        TEST.TST_P10S := TEST.TST_P10S + 1;
    END_IF;
    IF SYS.PLCCFG.PLS.P60S THEN
        TEST.TST_P60S := TEST.TST_P60S + 1;
    END_IF;
    IF SYS.PLCCFG.TQ - TEST.TEST_TQPREV >= 121 THEN
        TEST.TST_PLSON := false;
    END_IF;
ELSE
    TEST.TEST_TQPREV := SYS.PLCCFG.TQ;
END_IF;

IF SYS.PLCCFG.PLS.NEWHR THEN
    TEST.TST_CHHRCNT := TEST.TST_CHHRCNT + 1;
END_IF;
IF SYS.PLCCFG.PLS.NEWDAY THEN
    TEST.TST_CHDAYCNT := TEST.TST_CHDAYCNT + 1;
END_IF;

END_FUNCTION
